{attribute 'linkalways'} 
{attribute 'no_explicit_call' := 'This FB is a CLASS and must be accessed using methods or properties'}
{attribute 'enable_dynamic_creation'}
FUNCTION_BLOCK Node_ContainerType_Vector_TcVnVector2_REAL EXTENDS Node
VAR
    out : _GUID;
END_VAR

METHOD PUBLIC  Clone : I_Node
VAR
	pNode : POINTER TO Node_ContainerType_Vector_TcVnVector2_REAL;
END_VAR
pNode := __NEW(Node_ContainerType_Vector_TcVnVector2_REAL);
Clone := pNode^;
END_METHOD

METHOD FB_init : BOOL
VAR_INPUT
	bInitRetains : BOOL; // if TRUE, the retain variables are initialized (warm start / cold start)
	bInCopyCode : BOOL;  // if TRUE, the instance afterwards gets moved into the copy code (online change)
END_VAR
AddOutput('out', out);
END_METHOD

METHOD PROTECTED OnExecute
out.Value := ContainerType_Vector_TcVnVector2_REAL;
END_METHOD

END_FUNCTION_BLOCK

(* stored: Version 1.1.0.1, ProductVersion 3.1.4026.17
   POU Node_ContainerType_Vector_TcVnVector2_REAL: Id {aed48ef2-6564-02fd-36f7-2d1f92efdd98}, SpecialFunc None
   Folder Constructor: Id {28ccae8a-cc06-0c9e-3837-b913c16ca319}
   Method Clone: Id {cb59d59a-a6d2-0a5c-3339-51429966b0a8}
   Method FB_init: Id {b1f518cf-e020-020f-3671-577e48fbe2ce}
   Method OnExecute: Id {67415586-a017-0067-24d1-ef913185edd5} *)
